TYPE CT_Track_Tc_to_BR_t :
STRUCT
    bCommand : BYTE; (* command bit field for the track system *)
END_STRUCT
END_TYPE

(* stored: Version 1.1.0.1, ProductVersion 3.1.4024.6
   DUT CT_Track_Tc_to_BR_t: Id {f85518ed-8a0e-4ded-9191-92f3f24274ff} *)
